(* PLC project v0.6.02_RefactorGateAndTest.project, CODESYS CODESYS V3.5 SP19 Patch 1 *)
(* stored: creationDateTime 2026-08-14T10:10:49.391775, modificationDateTime 2026-08-14T10:10:49.391775 *)

TYPE ST_Winch_SymmetryCfg : STRUCT
  DeltaStartDelay_Ms : UDINT := 100;
  DeltaBrakeReleaseTime_Ms : UDINT := 100;
  DeltaBrakeApplyTime_Ms : UDINT := 100;
  DeltaStopDistance_Mm : UDINT := 100;
  DeltaStopTime_Ms : UDINT := 200;
  MinimumCommandTime_Ms : UDINT := 1000;
  MinimumSpeed_Mps : REAL := 0.05;
END_STRUCT;
END_TYPE
